// TIA Portal V18 export
TYPE "LGasp_type_Dati_Impilaggio"
// stored: IsFailsafeCompliant false
   STRUCT
      quota { ExternalVisible := 'False'; ExternalWritable := 'False'} : Array[1..200] of "LGasp_type_quote_impilaggio";
      Nr_pz_limitato_da_dimensioni { ExternalVisible := 'False'; ExternalWritable := 'False'} : Bool;   // Il calcolo dei numero di pezzi tot è limitato dalle dimensioni del pacco
      Nr_pz_limitato_da_peso { ExternalVisible := 'False'; ExternalWritable := 'False'} : Bool;   // Il calcolo dei numero di pezzi tot è limitato dal peso massimo del pacco
      Nr_pz_limitato_da_prog { ExternalVisible := 'False'; ExternalWritable := 'False'} : Bool;   // Il calcolo dei numero di pezzi tot è limitato dal programma
      N_righe_tot { ExternalVisible := 'False'; ExternalWritable := 'False'} : DInt;   // Numero di righe totali calcolate per pacco
      N_colonne_tot { ExternalVisible := 'False'; ExternalWritable := 'False'} : DInt;   // Numero di colonne totali calcolate per pacco
      N_Pezzi_tot : DInt;   // Numero di pezzi totali calcolati per pacco
      Peso_1pz { ExternalAccessible := 'False'; ExternalVisible := 'False'; ExternalWritable := 'False'} : LReal;   // [kg] peso singolo pezzo
   END_STRUCT;
END_TYPE
